// TIA Portal V17 export
// export: Created 2023-02-14T02:49:54.0093253Z, ExportSetting WithDefaults, DisplayName Totally Integrated Automation Portal, DisplayVersion V17, DisplayName TIA Portal Openness, DisplayVersion V17, DisplayName TIA Portal Teamcenter Gateway, DisplayVersion V17, DisplayName TIA Portal Version Control Interface, DisplayVersion V17, DisplayName SINAMICS Startdrive Advanced, DisplayVersion V17, DisplayName SINAMICS Startdrive G130, G150, S120, S150, SINAMICS MV, S210, DisplayVersion V17, DisplayName SINAMICS Startdrive G110M, G120, G120C, G120D, G120P, G115D, DisplayVersion V17, DisplayName STEP 7 Professional, DisplayVersion V17, DisplayName STEP 7 Safety, DisplayVersion V17, DisplayName WinCC Professional, DisplayVersion V17
VAR_GLOBAL   // PLC tag table "RIO Blending Panel"
   "ZSC-20.02" AT %I15.0 : Bool;
   "ZSC-20.03" AT %I15.1 : Bool;
   "ZSC-20.05" AT %I15.2 : Bool;
   "ZSC-20.06" AT %I15.3 : Bool;
   "ZSC-20.08" AT %I15.4 : Bool;
   "ZSC-20.09" AT %I15.5 : Bool;
   "ZSC-20.11" AT %I15.6 : Bool;
   "ZSC-20.21" AT %I15.7 : Bool;
   "ZSC-20.23" AT %I16.0 : Bool;
   "ZSC-20.24" AT %I16.1 : Bool;
   "ZSC-20.25" AT %I16.2 : Bool;
   "ZSC-20.27" AT %I16.3 : Bool;
   "ZSC-20.28" AT %I16.4 : Bool;
   "ZSC-20.31" AT %I16.5 : Bool;
   "ZSC-20.32" AT %I16.6 : Bool;
   "ZSC-20.33" AT %I16.7 : Bool;
   "ZSC-20.34" AT %I17.0 : Bool;
   "ZSC-20.35" AT %I17.1 : Bool;
   "ZSC-20.36" AT %I17.2 : Bool;
   "ZSC-20.37" AT %I17.3 : Bool;
   "ZSC-21.02" AT %I17.4 : Bool;
   "ZSC-21.03" AT %I17.5 : Bool;
   "ZSC-21.05" AT %I17.6 : Bool;
   "ZSC-21.06" AT %I17.7 : Bool;
   "ZSC-21.08" AT %I18.0 : Bool;
   "ZSC-21.09" AT %I18.1 : Bool;
   "ZSC-21.11" AT %I18.2 : Bool;
   "ZSC-21.21" AT %I18.3 : Bool;
   "ZSC-21.23" AT %I18.4 : Bool;
   "ZSC-21.24" AT %I18.5 : Bool;
   "ZSC-21.25" AT %I18.6 : Bool;
   "ZSC-21.27" AT %I18.7 : Bool;
   "ZSC-21.28" AT %I19.0 : Bool;
   "ZSC-21.31" AT %I19.1 : Bool;
   "ZSC-21.32" AT %I19.2 : Bool;
   "ZSC-21.33" AT %I19.3 : Bool;
   "ZSC-21.34" AT %I19.4 : Bool;
   "ZSC-21.35" AT %I19.5 : Bool;
   "ZSC-30.02" AT %I19.6 : Bool;
   "ZSC-30.03" AT %I19.7 : Bool;
   "ZSC-30.05" AT %I20.0 : Bool;
   "ZSC-30.06" AT %I20.1 : Bool;
   "ZSC-30.08" AT %I20.2 : Bool;
   "ZSC-30.09" AT %I20.3 : Bool;
   "ZSC-30.11" AT %I20.4 : Bool;
   "ZSC-30.14" AT %I20.5 : Bool;
   "ZSC-30.17" AT %I20.6 : Bool;
   "ZSC-30.20" AT %I20.7 : Bool;
   "ZSC-30.21" AT %I21.0 : Bool;
   "ZSC-30.23" AT %I21.1 : Bool;
   "ZSC-30.24" AT %I21.2 : Bool;
   "ZSC-30.25" AT %I21.3 : Bool;
   "ZSC-30.27" AT %I21.4 : Bool;
   "ZSC-30.28" AT %I21.5 : Bool;
   "ZSC-30.31" AT %I21.6 : Bool;
   "ZSC-30.32" AT %I21.7 : Bool;
   "ZSC-30.33" AT %I22.0 : Bool;
   "ZSC-30.34" AT %I22.1 : Bool;
   "ZSC-30.35" AT %I22.2 : Bool;
   "ZSC-30.36" AT %I22.3 : Bool;
   "spare blending" AT %I22.4 : Bool;
   "spare blending(1)" AT %I22.5 : Bool;
   "spare blending(2)" AT %I22.6 : Bool;
   "spare blending(3)" AT %I22.7 : Bool;
   "ZSC-31.02" AT %I23.0 : Bool;
   "ZSC-31.03" AT %I23.1 : Bool;
   "ZSC-31.05" AT %I23.2 : Bool;
   "ZSC-31.06" AT %I23.3 : Bool;
   "ZSC-31.08" AT %I23.4 : Bool;
   "ZSC-31.09" AT %I23.5 : Bool;
   "ZSC-31.11" AT %I23.6 : Bool;
   "ZSC-31.21" AT %I23.7 : Bool;
   "ZSC-31.23" AT %I24.0 : Bool;
   "ZSC-31.24" AT %I24.1 : Bool;
   "ZSC-31.25" AT %I24.2 : Bool;
   "ZSC-31.27" AT %I24.3 : Bool;
   "ZSC-31.28" AT %I24.4 : Bool;
   "ZSC-31.31" AT %I24.5 : Bool;
   "ZSC-31.32" AT %I24.6 : Bool;
   "ZSC-31.33" AT %I24.7 : Bool;
   "ZSC-31.34" AT %I25.0 : Bool;
   "ZSC-31.35" AT %I25.1 : Bool;
   "ZSC-40.02" AT %I25.2 : Bool;
   "ZSC-40.03" AT %I25.3 : Bool;
   "ZSC-40.05" AT %I25.4 : Bool;
   "ZSC-40.06" AT %I25.5 : Bool;
   "ZSC-40.08" AT %I25.6 : Bool;
   "ZSC-40.09" AT %I25.7 : Bool;
   "ZSC-40.11" AT %I26.0 : Bool;
   "ZSC-40.21" AT %I26.1 : Bool;
   "ZSC-40.23" AT %I26.2 : Bool;
   "ZSC-40.24" AT %I26.3 : Bool;
   "ZSC-40.25" AT %I26.4 : Bool;
   "ZSC-40.27" AT %I26.5 : Bool;
   "ZSC-40.28" AT %I26.6 : Bool;
   "ZSC-40.31" AT %I26.7 : Bool;
   "ZSC-40.32" AT %I27.0 : Bool;
   "ZSC-40.33" AT %I27.1 : Bool;
   "ZSC-40.34" AT %I27.2 : Bool;
   "ZSC-41.02" AT %I27.3 : Bool;
   "ZSC-41.03" AT %I27.4 : Bool;
   "ZSC-41.05" AT %I27.5 : Bool;
   "ZSC-41.06" AT %I27.6 : Bool;
   "ZSC-41.08" AT %I27.7 : Bool;
   "Pulse FT-00.01" AT %I28.0 : Bool;
   "PS-01" AT %I28.1 : Bool;
   "PS-02" AT %I28.2 : Bool;
   "PS-03" AT %I28.3 : Bool;
   "PS-04" AT %I28.4 : Bool;
   "spare blending(4)" AT %I28.5 : Bool;
   "spare blending(5)" AT %I28.6 : Bool;
   "spare blending(6)" AT %I28.7 : Bool;
   "Flowrate FT-00.01" AT %IW29 : Int;
   "LT-20.01" AT %IW31 : Int;
   "LT-21.01" AT %IW33 : Int;
   "LT-22.01" AT %IW35 : Int;
   "LT-30.01" AT %IW37 : Int;
   "LT-31.01" AT %IW39 : Int;
   "LT-32.01" AT %IW41 : Int;
   "LT-40.01" AT %IW43 : Int;
   "LT-41.01" AT %IW45 : Int;
   "spare blending(13)" AT %IW47 : Int;
   "spare blending(14)" AT %IW49 : Int;
   "spare blending(15)" AT %IW51 : Int;
   "ZSC-41.09" AT %I71.0 : Bool;
   "ZSC-41.11" AT %I71.1 : Bool;
   "ZSC-41.14" AT %I71.2 : Bool;
   "ZSC-41.17" AT %I71.3 : Bool;
   "ZSC-41.20" AT %I71.4 : Bool;
   "ZSC-41.21" AT %I71.5 : Bool;
   "ZSC-41.23" AT %I71.6 : Bool;
   "ZSC-41.24" AT %I71.7 : Bool;
   "ZSC-41.25" AT %I72.0 : Bool;
   "ZSC-41.27" AT %I72.1 : Bool;
   "ZSC-41.28" AT %I72.2 : Bool;
   "ZSC-41.31" AT %I72.3 : Bool;
   "ZSC-41.32" AT %I72.4 : Bool;
   "ZSC-41.33" AT %I72.5 : Bool;
   "ZSC-41.34" AT %I72.6 : Bool;
   "spare blending(16)" AT %I72.7 : Bool;
   "spare blending(17)" AT %I74.0 : Bool;
   "spare blending(18)" AT %I74.1 : Bool;
   "spare blending(19)" AT %I74.2 : Bool;
   "ZSC-61.01" AT %I74.3 : Bool;
   "ZSC-61.03" AT %I74.4 : Bool;
   "spare blending(20)" AT %I74.5 : Bool;
   "spare blending(21)" AT %I74.6 : Bool;
   "ZSC-62.06" AT %I74.7 : Bool;
   "spare blending(22)" AT %I892.0 : Bool;
   "spare blending(23)" AT %I892.1 : Bool;
   "ZSC-64.01" AT %I892.2 : Bool;
   "ZSC-64.03" AT %I892.3 : Bool;
   "ZSC-64.06" AT %I892.4 : Bool;
   "ZSC-65.01" AT %I892.5 : Bool;
   "ZSC-65.03" AT %I892.6 : Bool;
   "ZSC-66.01" AT %I892.7 : Bool;
   "ZSC-66.03" AT %I893.0 : Bool;
   "ZSC-66.06" AT %I893.1 : Bool;
   "ZSC-67.01" AT %I893.2 : Bool;
   "ZSC-67.03" AT %I893.3 : Bool;
   "ZSC-68.01" AT %I893.4 : Bool;
   "ZSC-68.03" AT %I893.5 : Bool;
   "ZSC-68.06" AT %I893.6 : Bool;
   "EM STOP RIO BLENDING" AT %I893.7 : Bool;
   "DRP-P22.01" AT %I894.0 : Bool;
   "DRP-P32.01" AT %I894.1 : Bool;
   "spare blending(24)" AT %I894.2 : Bool;
   "spare blending(25)" AT %I894.3 : Bool;
   "spare blending(26)" AT %I894.4 : Bool;
   "spare blending(27)" AT %I894.5 : Bool;
   "spare blending(28)" AT %I894.6 : Bool;
   "spare blending(29)" AT %I894.7 : Bool;
   "DRP-P22.01 Switching Input" AT %Q3.0 : Bool;
   "DRP-P32.01 Switching Input" AT %Q3.1 : Bool;
   "spare blending(7)" AT %Q3.2 : Bool;
   "spare blending(8)" AT %Q3.3 : Bool;
   "spare blending(9)" AT %Q3.4 : Bool;
   "spare blending(10)" AT %Q3.5 : Bool;
   "spare blending(11)" AT %Q3.6 : Bool;
   "spare blending(12)" AT %Q3.7 : Bool;
   "AV-20.01" AT %Q26.0 : Bool;
   "AV-20.02" AT %Q26.1 : Bool;
   "AV-20.03" AT %Q26.2 : Bool;
   "AV-20.04" AT %Q26.3 : Bool;
   "AV-20.05" AT %Q26.4 : Bool;
   "AV-20.06" AT %Q26.5 : Bool;
   "AV-20.07" AT %Q26.6 : Bool;
   "AV-20.08" AT %Q26.7 : Bool;
   "AV-20.09" AT %Q27.0 : Bool;
   "AV-20.10" AT %Q27.1 : Bool;
   "AV-20.11" AT %Q27.2 : Bool;
   "AV-20.21" AT %Q27.3 : Bool;
   "AV-20.22" AT %Q27.4 : Bool;
   "AV-20.23" AT %Q27.5 : Bool;
   "AV-20.24" AT %Q27.6 : Bool;
   "AV-20.25" AT %Q27.7 : Bool;
   "AV-20.26" AT %Q28.0 : Bool;
   "AV-20.27" AT %Q28.1 : Bool;
   "AV-20.28" AT %Q28.2 : Bool;
   "AV-20.29" AT %Q28.3 : Bool;
   "AV-20.30" AT %Q28.4 : Bool;
   "AV-20.31" AT %Q28.5 : Bool;
   "AV-20.32" AT %Q28.6 : Bool;
   "AV-20.33" AT %Q28.7 : Bool;
   "AV-20.34" AT %Q29.0 : Bool;
   "AV-20.35" AT %Q29.1 : Bool;
   "AV-20.36" AT %Q29.2 : Bool;
   "AV-20.37" AT %Q29.3 : Bool;
   "AV-20.41" AT %Q29.4 : Bool;
   "AV-20.42" AT %Q29.5 : Bool;
   "AV-21.01" AT %Q29.6 : Bool;
   "AV-21.02" AT %Q29.7 : Bool;
   "AV-21.03" AT %Q30.0 : Bool;
   "AV-21.04" AT %Q30.1 : Bool;
   "AV-21.05" AT %Q30.2 : Bool;
   "AV-21.06" AT %Q30.3 : Bool;
   "AV-21.07" AT %Q30.4 : Bool;
   "AV-21.08" AT %Q30.5 : Bool;
   "AV-21.09" AT %Q30.6 : Bool;
   "AV-21.10" AT %Q30.7 : Bool;
   "AV-21.11" AT %Q31.0 : Bool;
   "AV-21.21" AT %Q31.1 : Bool;
   "AV-21.22" AT %Q31.2 : Bool;
   "AV-21.23" AT %Q31.3 : Bool;
   "AV-21.24" AT %Q31.4 : Bool;
   "AV-21.25" AT %Q31.5 : Bool;
   "AV-21.26" AT %Q31.6 : Bool;
   "AV-21.27" AT %Q31.7 : Bool;
   "AV-21.28" AT %Q32.0 : Bool;
   "AV-21.29" AT %Q32.1 : Bool;
   "AV-21.30" AT %Q32.2 : Bool;
   "AV-21.31" AT %Q32.3 : Bool;
   "AV-21.32" AT %Q32.4 : Bool;
   "AV-21.33" AT %Q32.5 : Bool;
   "AV-21.34" AT %Q32.6 : Bool;
   "AV-21.35" AT %Q32.7 : Bool;
   "AV-21.41" AT %Q33.0 : Bool;
   "AV-21.42" AT %Q33.1 : Bool;
   "AV-30.01" AT %Q33.2 : Bool;
   "AV-30.02" AT %Q33.3 : Bool;
   "AV-30.03" AT %Q33.4 : Bool;
   "AV-30.04" AT %Q33.5 : Bool;
   "AV-30.05" AT %Q33.6 : Bool;
   "AV-30.06" AT %Q33.7 : Bool;
   "AV-30.07" AT %Q34.0 : Bool;
   "AV-30.08" AT %Q34.1 : Bool;
   "AV-30.09" AT %Q34.2 : Bool;
   "AV-30.10" AT %Q34.3 : Bool;
   "AV-30.11" AT %Q34.4 : Bool;
   "AV-30.12" AT %Q34.5 : Bool;
   "AV-30.13" AT %Q34.6 : Bool;
   "AV-30.14" AT %Q34.7 : Bool;
   "AV-30.15" AT %Q35.0 : Bool;
   "AV-30.16" AT %Q35.1 : Bool;
   "AV-30.17" AT %Q35.2 : Bool;
   "AV-30.18" AT %Q35.3 : Bool;
   "AV-30.19" AT %Q35.4 : Bool;
   "AV-30.20" AT %Q35.5 : Bool;
   "AV-30.21" AT %Q35.6 : Bool;
   "AV-30.22" AT %Q35.7 : Bool;
   "AV-30.23" AT %Q36.0 : Bool;
   "AV-30.24" AT %Q36.1 : Bool;
   "AV-30.25" AT %Q36.2 : Bool;
   "AV-30.26" AT %Q36.3 : Bool;
   "AV-30.27" AT %Q36.4 : Bool;
   "AV-30.28" AT %Q36.5 : Bool;
   "AV-30.29" AT %Q36.6 : Bool;
   "AV-30.30" AT %Q36.7 : Bool;
   "AV-30.31" AT %Q37.0 : Bool;
   "AV-30.32" AT %Q37.1 : Bool;
   "AV-30.33" AT %Q37.2 : Bool;
   "AV-30.34" AT %Q37.3 : Bool;
   "AV-30.35" AT %Q37.4 : Bool;
   "AV-30.36" AT %Q37.5 : Bool;
   "AV-30.41" AT %Q37.6 : Bool;
   "AV-30.42" AT %Q37.7 : Bool;
   "AV-22.11" AT %Q38.5 : Bool;
   "AV-22.21" AT %Q38.6 : Bool;
   "AV-22.22" AT %Q38.7 : Bool;
   "AV-22.23" AT %Q39.0 : Bool;
   "AV-31.01" AT %Q39.1 : Bool;
   "AV-31.02" AT %Q39.2 : Bool;
   "AV-31.03" AT %Q39.3 : Bool;
   "AV-31.04" AT %Q39.4 : Bool;
   "AV-31.05" AT %Q39.5 : Bool;
   "AV-31.06" AT %Q39.6 : Bool;
   "AV-31.07" AT %Q39.7 : Bool;
   "AV-31.08" AT %Q40.0 : Bool;
   "AV-31.09" AT %Q40.1 : Bool;
   "AV-31.10" AT %Q40.2 : Bool;
   "AV-31.11" AT %Q40.3 : Bool;
   "AV-31.21" AT %Q40.4 : Bool;
   "AV-31.22" AT %Q40.5 : Bool;
   "AV-31.23" AT %Q40.6 : Bool;
   "AV-31.24" AT %Q40.7 : Bool;
   "AV-31.25" AT %Q41.0 : Bool;
   "AV-31.26" AT %Q41.1 : Bool;
   "AV-31.27" AT %Q41.2 : Bool;
   "AV-31.28" AT %Q41.3 : Bool;
   "AV-31.29" AT %Q41.4 : Bool;
   "AV-31.30" AT %Q41.5 : Bool;
   "AV-31.31" AT %Q41.6 : Bool;
   "AV-31.32" AT %Q41.7 : Bool;
   "AV-31.33" AT %Q42.0 : Bool;
   "AV-31.34" AT %Q42.1 : Bool;
   "AV-31.35" AT %Q42.2 : Bool;
   "AV-31.41" AT %Q42.3 : Bool;
   "AV-31.42" AT %Q42.4 : Bool;
   "AV-40.01" AT %Q42.5 : Bool;
   "AV-40.02" AT %Q42.6 : Bool;
   "AV-40.03" AT %Q42.7 : Bool;
   "AV-40.04" AT %Q43.0 : Bool;
   "AV-40.05" AT %Q43.1 : Bool;
   "AV-40.06" AT %Q43.2 : Bool;
   "AV-40.07" AT %Q43.3 : Bool;
   "AV-40.08" AT %Q43.4 : Bool;
   "AV-40.09" AT %Q43.5 : Bool;
   "AV-40.10" AT %Q43.6 : Bool;
   "AV-40.11" AT %Q43.7 : Bool;
   "AV-40.21" AT %Q44.0 : Bool;
   "AV-40.22" AT %Q44.1 : Bool;
   "AV-40.23" AT %Q44.2 : Bool;
   "AV-40.24" AT %Q44.3 : Bool;
   "AV-40.25" AT %Q110.0 : Bool;
   "AV-40.26" AT %Q110.1 : Bool;
   "AV-40.27" AT %Q110.2 : Bool;
   "AV-40.28" AT %Q110.3 : Bool;
   "AV-40.29" AT %Q110.4 : Bool;
   "AV-40.30" AT %Q110.5 : Bool;
   "AV-40.31" AT %Q110.6 : Bool;
   "AV-40.32" AT %Q110.7 : Bool;
   "AV-40.33" AT %Q111.0 : Bool;
   "AV-40.34" AT %Q111.1 : Bool;
   "AV-41.01" AT %Q111.2 : Bool;
   "AV-41.02" AT %Q111.3 : Bool;
   "AV-41.03" AT %Q111.4 : Bool;
   "AV-41.04" AT %Q111.5 : Bool;
   "AV-41.05" AT %Q111.6 : Bool;
   "AV-41.06" AT %Q111.7 : Bool;
   "AV-41.07" AT %Q112.0 : Bool;
   "AV-41.08" AT %Q112.1 : Bool;
   "AV-41.09" AT %Q112.2 : Bool;
   "AV-41.10" AT %Q112.3 : Bool;
   "AV-41.11" AT %Q112.4 : Bool;
   "AV-41.12" AT %Q112.5 : Bool;
   "AV-41.13" AT %Q112.6 : Bool;
   "AV-41.14" AT %Q112.7 : Bool;
   "AV-41.15" AT %Q113.0 : Bool;
   "AV-41.16" AT %Q113.1 : Bool;
   "AV-41.17" AT %Q113.2 : Bool;
   "AV-41.18" AT %Q113.3 : Bool;
   "AV-41.19" AT %Q113.4 : Bool;
   "AV-41.20" AT %Q113.5 : Bool;
   "AV-41.21" AT %Q113.6 : Bool;
   "AV-41.22" AT %Q113.7 : Bool;
   "AV-41.23" AT %Q114.0 : Bool;
   "AV-41.24" AT %Q114.1 : Bool;
   "AV-41.25" AT %Q114.2 : Bool;
   "AV-41.26" AT %Q114.3 : Bool;
   "AV-41.27" AT %Q114.4 : Bool;
   "AV-41.28" AT %Q114.5 : Bool;
   "AV-41.29" AT %Q114.6 : Bool;
   "AV-41.30" AT %Q114.7 : Bool;
   "AV-41.31" AT %Q115.0 : Bool;
   "AV-41.32" AT %Q115.1 : Bool;
   "AV-41.33" AT %Q115.2 : Bool;
   "AV-41.34" AT %Q115.3 : Bool;
   "AV-32.01" AT %Q115.4 : Bool;
   "AV-32.02" AT %Q115.5 : Bool;
   "AV-32.03" AT %Q115.6 : Bool;
   "AV-32.04" AT %Q115.7 : Bool;
   "AV-32.11" AT %Q90.1 : Bool;
   "AV-32.21" AT %Q90.2 : Bool;
   "AV-32.22" AT %Q90.3 : Bool;
   "AV-32.23" AT %Q90.4 : Bool;
   "AV-61.01" AT %Q90.5 : Bool;
   "AV-61.02" AT %Q90.6 : Bool;
   "AV-61.03" AT %Q90.7 : Bool;
   "AV-61.04" AT %Q91.0 : Bool;
   "AV-61.05" AT %Q91.1 : Bool;
   "AV-61.21" AT %Q91.2 : Bool;
   "AV-62.06" AT %Q92.0 : Bool;
   "AV-64.01" AT %Q92.6 : Bool;
   "AV-64.02" AT %Q92.7 : Bool;
   "AV-64.03" AT %Q93.0 : Bool;
   "AV-64.04" AT %Q93.1 : Bool;
   "AV-64.05" AT %Q93.2 : Bool;
   "AV-64.06" AT %Q93.3 : Bool;
   "Av-65.01" AT %Q93.4 : Bool;
   "Av-65.02" AT %Q93.5 : Bool;
   "Av-65.03" AT %Q93.6 : Bool;
   "Av-65.04" AT %Q93.7 : Bool;
   "AV-65.05" AT %Q94.0 : Bool;
   "AV-65.21" AT %Q94.1 : Bool;
   "AV-66.01" AT %Q94.2 : Bool;
   "AV-66.02" AT %Q94.3 : Bool;
   "AV-66.03" AT %Q94.4 : Bool;
   "AV-66.04" AT %Q94.5 : Bool;
   "AV-66.05" AT %Q94.6 : Bool;
   "AV-66.06" AT %Q94.7 : Bool;
   "AV-67.01" AT %Q95.0 : Bool;
   "AV-67.02" AT %Q95.1 : Bool;
   "AV-67.03" AT %Q95.2 : Bool;
   "AV-67.04" AT %Q95.3 : Bool;
   "AV-67.05" AT %Q95.4 : Bool;
   "AV-68.01" AT %Q95.5 : Bool;
   "AV-68.02" AT %Q95.6 : Bool;
   "AV-68.03" AT %Q95.7 : Bool;
   "AV-68.04" AT %Q96.0 : Bool;
   "AV-68.05" AT %Q96.1 : Bool;
   "AV-68.06" AT %Q96.2 : Bool;
END_VAR
